Omron Sysmac Studio project Matching_Code_10 (Sysmac Studio 1.54.0.64019, StandardProject)
(* update 6_7 / have modify the res for fully reset home flag *)

# Controller new_Controller_0: NX1P2-1140DT version 1.18
Units and slaves: Node47 : MADLN05BE (E002); Node72 : MADLN05BE (E001); Node73 : MADLN05BE (E003)
Axis MC_Axis1, settings changed from default: AxisType=ServoType, UnitsConversion=EnumElement5, UnitsNumerator=8388608, UnitsDenominator=36, MaxVelocity=500, MaxJogVelocity=360, SoftwareLimitMode=ValidForSpecifiedValueImmediateStop, PositiveSoftwareLimit=75, NegativeSoftwareLimit=-29.2, OriginInputMode=EXT, StartDirection=NegativeDirection, OriginInputDetectionDirection=NegativeDirection, HomingVelocity=100, HomingApproachVelocity=10, HomingAcceleration=10, HomingDeceleration=20
Axis MC_Axis2, settings changed from default: AxisNumber=1, AxisType=ServoType, UnitsConversion=EnumElement5, UnitsNumerator=8388608, UnitsDenominator=36, MaxVelocity=500, MaxJogVelocity=360, SoftwareLimitMode=ValidForSpecifiedValueImmediateStop, PositiveSoftwareLimit=75, NegativeSoftwareLimit=-29.2
Axis MC_Axis3, settings changed from default: AxisNumber=2, AxisType=ServoType, UnitsConversion=EnumElement5, UnitsNumerator=8388608, UnitsDenominator=36, MaxVelocity=500, MaxJogVelocity=360, SoftwareLimitMode=ValidForSpecifiedValueDecreaseStop, PositiveSoftwareLimit=29.2, NegativeSoftwareLimit=-75
Task PrimaryTask (priority 4, period or condition 4000): Program0

TYPE InforRobot : STRUCT
    e : LREAL;
    rf : LREAL;
    re : LREAL;
    f : LREAL;
END_STRUCT END_TYPE
TYPE Input_Position : STRUCT
    X : LREAL;
    Y : LREAL;
    Z : LREAL;
END_STRUCT END_TYPE
TYPE Angle_Theta : STRUCT
    Theta1 : LREAL;
    Theta2 : LREAL;
    Theta3 : LREAL;
END_STRUCT END_TYPE
TYPE Bool_Theta : STRUCT
    Motor_Theta1 : REAL;
    Motor_Theta2 : REAL;
    Motor_Theta3 : REAL;
END_STRUCT END_TYPE
TYPE Speed_Theta : STRUCT
    Speed_Theta1 : REAL;
    Speed_Theta2 : REAL;
    Speed_Theta3 : REAL;
END_STRUCT END_TYPE
TYPE Workspace : STRUCT
    X_Min : REAL;
    X_Max : REAL;
    Y_Min : REAL;
    Y_Max : REAL;
    Z_Min : REAL;
    Z_Max : REAL;
END_STRUCT END_TYPE
TYPE From_pc : STRUCT
    commandID : INT;
    argument_number : INT;
    argument_x : ARRAY[0..6] OF real;
    argument_y : ARRAY[0..6] OF real;
    argument_z : ARRAY[0..6] OF real;
    argument_time : ARRAY[0..6] OF real;
    argument_e : ARRAY[0..6] OF int;
    bit_doing : INT;
END_STRUCT END_TYPE
TYPE From_plc : STRUCT
    pos_angular : ARRAY[0..2] OF REAL;
    pos_EE : ARRAY[0..6] OF REAL;
    task_doing : INT;
    task_state : INT;
    Total_Time_Estimate : ARRAY[0..6] OF REAL;
END_STRUCT END_TYPE

VAR_GLOBAL CONSTANT
    MC_Axis1 : _sAXIS_REF;  (* at MC://_MC_AX[0] *)
    MC_Axis2 : _sAXIS_REF;  (* at MC://_MC_AX[1] *)
    MC_Axis3 : _sAXIS_REF;  (* at MC://_MC_AX[2] *)
END_VAR
VAR_GLOBAL
    Out_Test0 : LREAL;
    Out_TestAngle1 : LREAL;
    Out_TestAngle2 : LREAL;
    Out_TestAngle3 : LREAL;
    MyHomingPara : _sHOMING_REF;
    Home_Axis1 : BOOL;  (* at BuiltInIO://cpu/#0/Input_Bit_00 *)
    Home_Axis2 : BOOL;  (* at BuiltInIO://cpu/#0/Input_Bit_01 *)
    Home_Axis3 : BOOL;  (* at BuiltInIO://cpu/#0/Input_Bit_02 *)
    Home_Lamp1 : BOOL;  (* at BuiltInIO://cpu/#0/Output_Bit_00 *)
    Home_Lamp2 : BOOL;  (* at BuiltInIO://cpu/#0/Output_Bit_01 *)
    Home_Lamp3 : BOOL;  (* at BuiltInIO://cpu/#0/Output_Bit_02 *)
    Out_Done_Inter : BOOL;
    pc_package : From_pc;  (* published *)
    plc_package : From_plc;  (* published *)
    Pump_Out : BOOL;  (* at BuiltInIO://cpu/#0/Output_Bit_03 *)
    Mc_On_Btn : BOOL;  (* at BuiltInIO://cpu/#0/Input_Bit_03 *)
    Res_Err_Btn : BOOL;  (* at BuiltInIO://cpu/#0/Input_Bit_04 *)
    Valve_Out : BOOL;  (* at BuiltInIO://cpu/#0/Output_Bit_04 *)
    ICV_t : ARRAY[0..6] OF Lreal;
    Start_Home_Flag : BOOL;
    Home_Done_Flag1 : BOOL;
    Home_Done_Flag2 : BOOL;
    Home_Done_Flag3 : BOOL;
END_VAR

PROGRAM Program0
VAR
    Pw_servo_on : BOOL := False;
    MC_Move_Abs : BOOL;
    Pw_Power_0 : MC_Power;
    Pw_Power_1 : MC_Power;
    Pw_Power_2 : MC_Power;
    MC_Home_Ext : BOOL;  (* toggle 1 *)
    MC_Home_Delta_0 : MC_Home_Delta;
    Calib_Abs1 : MC_MoveAbsolute;
    Calib_Abs2 : MC_MoveAbsolute;
    Calib_Abs3 : MC_MoveAbsolute;
    Home_test_1 : MC_Home;
    Home_test_2 : MC_Home;
    Home_test_3 : MC_Home;
    Move_abs_0 : MC_MoveAbsolute;
    Move_abs_1 : MC_MoveAbsolute;
    Move_abs_2 : MC_MoveAbsolute;
    X_cal : LREAL;
    Y_cal : LREAL;
    Z_cal : LREAL;
    pos_angular : LREAL;
    Exe_Inter1 : BOOL;
    Exe_Inter2 : BOOL;
    Count1 : UINT;
    Count2 : UINT;
    Goto_Abs : Goto_Absolute;
    when_it_turn2 : BOOL;
    Goto_abs_x : LREAL;
    Goto_abs_y : LREAL;
    Goto_abs_z : LREAL;
    another3 : BOOL;
    Count3 : UINT;
    another4 : BOOL;
    Count4 : UINT;
    MC_Inter_Curve_Vel_0 : MC_Inter_Curve_Vel;
    MC_Inter_Curve_Vel_1 : MC_Inter_Curve_Vel;
    MC_Inter_Curve_Vel_2 : MC_Inter_Curve_Vel;
    MC_Inter_Curve_Vel_3 : MC_Inter_Curve_Vel;
    MC_Inter_Curve_Vel_4 : MC_Inter_Curve_Vel;
    MC_Inter_Curve_Vel_5 : MC_Inter_Curve_Vel;
    ICV_Start_NewTurn : BOOL;  (* Set 1 until ICV_Blend_done_2 *)
    ICV_Blend_Done_0 : BOOL;  (* Exe auto turn zero right after finish the blend, and blend will true right after *)
    ICV_Blend_Done_1 : BOOL;
    ICV_Blend_Done_2 : BOOL;
    ICV_Blend_Done_3 : BOOL;
    ICV_Blend_Done_4 : BOOL;
    ICV_Blend_Done_5 : BOOL;
    ICV_Vend_0 : LREAL;  (* Err_IK must reset manual *)
    ICV_Vend_1 : LREAL;
    ICV_Vend_2 : LREAL;
    ICV_Vend_3 : LREAL;
    ICV_Vend_4 : LREAL;
    ICV_Vend_5 : LREAL;
    ICV_Vmax : LREAL := 300;  (* 300 *)
    ICV_Amax : LREAL := 1000;  (* 1000 *)
    ICV_Dmax : LREAL := 1000;  (* 1000 *)
    Pump_Ext : BOOL;
    ICV_Pos_E : ARRAY[0..6] OF Int;
    ICV_Pos_X : ARRAY[0..6] OF Lreal;
    ICV_Pos_Y : ARRAY[0..6] OF Lreal;
    ICV_Pos_Z : ARRAY[0..6] OF Lreal;
    i1 : INT;
    MC_Goto_Abs : BOOL;  (* Set 1 until it done *)
    Fwk_Calc_OutX : REAL;
    Fwk_Calc_OutY : REAL;
    Fwk_Calc_OutZ : REAL;
    Moveto_Intermediary : MC_MoveAbsolute;
    Moveto_Midpoint : MC_MoveAbsolute;
    Moveto_Midpoint_1 : MC_MoveAbsolute;
    Moveto_Midpoint_2 : MC_MoveAbsolute;
    Moveto_Midpoint_3 : MC_MoveAbsolute;
    Home_Done : BOOL;
    Home_Error : BOOL;
    Goto_Abs_Error : BOOL;
    Pump_Res : BOOL;
    MC_ICV_Err : BOOL;
    MC_Stop1 : MC_Stop;
    MC_Stop2 : MC_Stop;
    MC_Stop3 : MC_Stop;
    MC_RES_DB1 : MC_Reset;
    MC_RES_DB2 : MC_Reset;
    MC_RES_DB3 : MC_Reset;
    Comment : BOOL;
    Mc_On_Btn_Flag : BOOL;
    Check_IK : BOOL;
    Goto_Abs2 : Goto_Absolute;
    Goto_Abs2_Exe : BOOL;
    Goto_Abs2_Done : BOOL;
    Out_TestAngle1_tmp : LREAL;
    Out_TestAngle2_tmp : LREAL;
    Out_TestAngle3_tmp : LREAL;
    Out_TestAngle10 : LREAL;
    Out_TestAngle20 : LREAL;
    Out_TestAngle30 : LREAL;
    Stop1 : MC_Power;
    MC_Stop4 : MC_Stop;
    MC_Stop5 : MC_Stop;
    MC_Stop6 : MC_Stop;
    Comment0 : BOOL;
    MC_Inter_Curve_Vel_6 : MC_Inter_Curve_Vel;
    ICV_Blend_Done_6 : BOOL;
    ICV_Vend_6 : LREAL;
    Current_Step : INT;
    Axis1_test : LREAL;
    Axis2_test : LREAL;
    Axis3_test : LREAL;
    fb_PumpTimer : TP;
    Var_Timer_IN : BOOL;
    ICV_t0 : LREAL;
    ICV_t1 : LREAL;
    ICV_t2 : LREAL;
    ICV_t3 : LREAL;
    ICV_t4 : LREAL;
    ICV_t5 : LREAL;
    Timing_for_EEF : TIME;
    i_t : INT;
    Mem_ICV_t5 : LREAL;
    k_t : LREAL;
    Pos_calib1 : LREAL;
    Pos_calib2 : LREAL;
    Pos_calib3 : LREAL;
END_VAR
VAR_EXTERNAL
    Out_Test0 : LREAL;
    Out_TestAngle1 : LREAL;
    Out_TestAngle2 : LREAL;
    Out_TestAngle3 : LREAL;
END_VAR
VAR_EXTERNAL CONSTANT
    MC_Axis1 : _sAXIS_REF;
    MC_Axis2 : _sAXIS_REF;
    MC_Axis3 : _sAXIS_REF;
END_VAR
VAR_EXTERNAL
    Home_Axis2 : BOOL;
    Home_Axis3 : BOOL;
    Out_Done_Inter : BOOL;
    plc_package : From_plc;
    pc_package : From_pc;
    Pump_Out : BOOL;
    Home_Axis1 : BOOL;
    Mc_On_Btn : BOOL;
    Res_Err_Btn : BOOL;
    Valve_Out : BOOL;
    ICV_t : ARRAY[0..6] OF Lreal;
    Start_Home_Flag : BOOL;
    Home_Done_Flag1 : BOOL;
    Home_Done_Flag2 : BOOL;
    Home_Done_Flag3 : BOOL;
END_VAR
VAR
    _p1 : BOOL;
    _t2 : BOOL;
    _t3 : BOOL;
END_VAR

(* Section Section0: ladder, written here as Structured Text *)

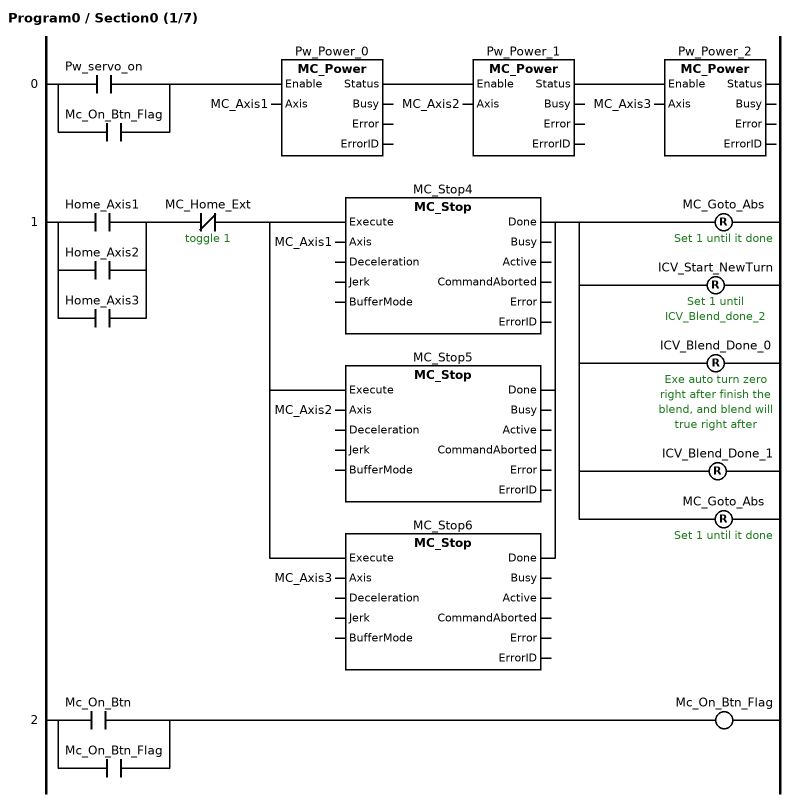
(* Rung 0 *)
Pw_Power_0(Enable := Pw_servo_on OR Mc_On_Btn_Flag, Axis := MC_Axis1);
Pw_Power_1(Enable := Pw_Power_0.Status, Axis := MC_Axis2);
Pw_Power_2(Enable := Pw_Power_1.Status, Axis := MC_Axis3);
(* Rung 1 *)
_p1 := (Home_Axis1 OR Home_Axis2 OR Home_Axis3) AND NOT MC_Home_Ext;
MC_Stop4(Execute := _p1, Axis := MC_Axis1);
MC_Stop5(Execute := _p1, Axis := MC_Axis2);
MC_Stop6(Execute := _p1, Axis := MC_Axis3);
IF MC_Stop4.Done OR MC_Stop5.Done OR MC_Stop6.Done THEN
    MC_Goto_Abs := FALSE;
    ICV_Start_NewTurn := FALSE;
    ICV_Blend_Done_0 := FALSE;
    ICV_Blend_Done_1 := FALSE;
    MC_Goto_Abs := FALSE;
END_IF;
(* Rung 2 *)
Mc_On_Btn_Flag := Mc_On_Btn OR Mc_On_Btn_Flag;

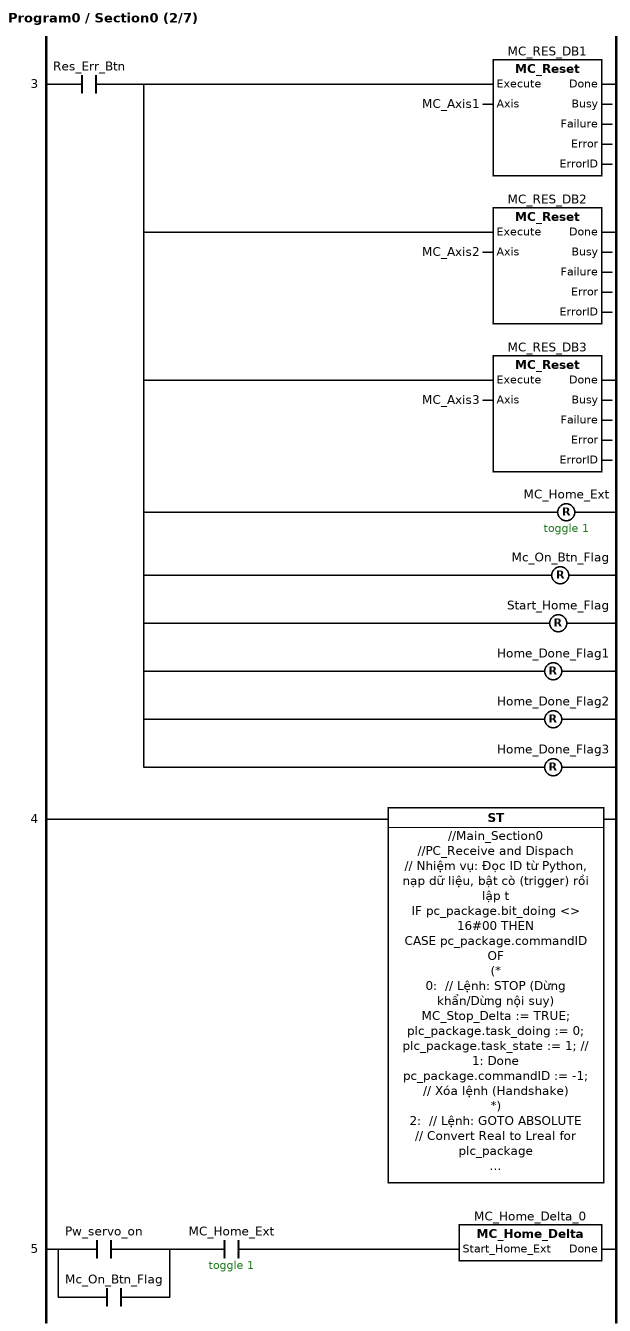
(* Rung 3 *)
MC_RES_DB1(Execute := Res_Err_Btn, Axis := MC_Axis1);
MC_RES_DB2(Execute := Res_Err_Btn, Axis := MC_Axis2);
MC_RES_DB3(Execute := Res_Err_Btn, Axis := MC_Axis3);
IF Res_Err_Btn THEN
    MC_Home_Ext := FALSE;
    Mc_On_Btn_Flag := FALSE;
    Start_Home_Flag := FALSE;
    Home_Done_Flag1 := FALSE;
    Home_Done_Flag2 := FALSE;
    Home_Done_Flag3 := FALSE;
END_IF;
(* Rung 4 *)
//Main_Section0 
//PC_Receive and Dispach
// Nhiệm vụ: Đọc ID từ Python, nạp dữ liệu, bật cò (trigger) rồi lập tức xóa ID

IF pc_package.bit_doing <> 16#00 THEN
CASE pc_package.commandID OF
  (*  
0:  // Lệnh: STOP (Dừng khẩn/Dừng nội suy)
	        MC_Stop_Delta := TRUE;
	        
	        plc_package.task_doing := 0;
	        plc_package.task_state := 1; // 1: Done
	        pc_package.commandID := -1;  // Xóa lệnh (Handshake)
			*)
    2:  // Lệnh: GOTO ABSOLUTE
		// Convert Real to Lreal for plc_package
		Goto_abs_x:= REAL_TO_LREAL(pc_package.argument_x[0]);
		Goto_abs_y := REAL_TO_LREAL(pc_package.argument_y[0]);
		Goto_abs_z:= REAL_TO_LREAL(pc_package.argument_z[0]);
        
        MC_Goto_Abs := TRUE;         // Bật cò chạy
        plc_package.task_doing := 2;
        plc_package.task_state := 2; // 2: Busy
        pc_package.commandID := -1;

    3:  // Lệnh: GO TRAJECTORY (Chạy quỹ đạo theo mảng tọa độ)
        ICV_Start_NewTurn := TRUE; //auto turn off
        FOR i1 := 0 TO 6 DO
			ICV_Pos_X[i1] := REAL_TO_LREAL(pc_package.argument_x[i1]);
			ICV_Pos_Y[i1] := REAL_TO_LREAL(pc_package.argument_y[i1]);
			ICV_Pos_Z[i1] := REAL_TO_LREAL(pc_package.argument_z[i1]);
			ICV_Pos_E[i1] := pc_package.argument_e[i1];
		END_FOR;
        plc_package.task_doing := 3;
        plc_package.task_state := 2; // Busy
        pc_package.commandID := -1;

    4:  // Lệnh: HOME CALIBRATION (Tìm gốc)
        MC_Home_Ext := TRUE;
        
        plc_package.task_doing := 4;
        plc_package.task_state := 2; // Busy
        pc_package.commandID := -1;

    5:  // Lệnh: PICK (Hút vật)
        Pump_Ext := TRUE;
        
        plc_package.task_doing := 5;
        plc_package.task_state := 1; // 1: Done (Do bật bơm là xong ngay)
        pc_package.commandID := -1;

    6:  // Lệnh: RELEASE (Nhả vật)
        Pump_Ext := FALSE;
        
        plc_package.task_doing := 6;
        plc_package.task_state := 1; // Done
        pc_package.commandID := -1;
		END_CASE;
pc_package.bit_doing :=16#00;
END_IF;
(* Rung 5 *)
MC_Home_Delta_0(Start_Home_Ext := (Pw_servo_on OR Mc_On_Btn_Flag) AND MC_Home_Ext);

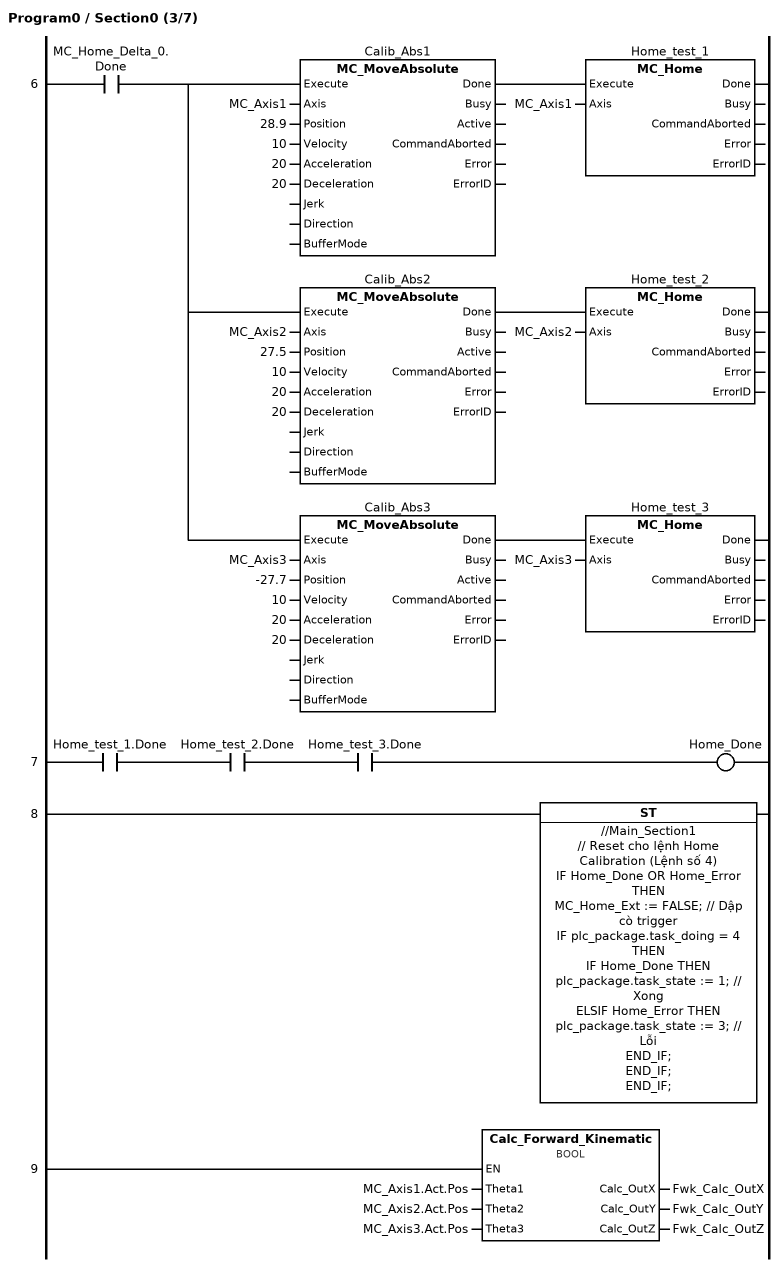
(* Rung 6 *)
Calib_Abs1(Execute := MC_Home_Delta_0.Done, Axis := MC_Axis1, Position := 28.9, Velocity := 10, Acceleration := 20, Deceleration := 20);
Home_test_1(Execute := Calib_Abs1.Done, Axis := MC_Axis1);
Calib_Abs2(Execute := MC_Home_Delta_0.Done, Axis := MC_Axis2, Position := 27.5, Velocity := 10, Acceleration := 20, Deceleration := 20);
Home_test_2(Execute := Calib_Abs2.Done, Axis := MC_Axis2);
Calib_Abs3(Execute := MC_Home_Delta_0.Done, Axis := MC_Axis3, Position := -27.7, Velocity := 10, Acceleration := 20, Deceleration := 20);
Home_test_3(Execute := Calib_Abs3.Done, Axis := MC_Axis3);
(* Rung 7 *)
Home_Done := Home_test_1.Done AND Home_test_2.Done AND Home_test_3.Done;
(* Rung 8 *)
//Main_Section1 
// Reset cho lệnh Home Calibration (Lệnh số 4)
IF Home_Done OR Home_Error THEN
 
    MC_Home_Ext := FALSE; // Dập cò trigger
	
    IF plc_package.task_doing = 4 THEN
        IF Home_Done THEN
            plc_package.task_state := 1; // Xong
        ELSIF Home_Error THEN
            plc_package.task_state := 3; // Lỗi
        END_IF;
    END_IF;
    
END_IF;
(* Rung 9 *)
_t2 := Calc_Forward_Kinematic(Theta1 := MC_Axis1.Act.Pos, Theta2 := MC_Axis2.Act.Pos, Theta3 := MC_Axis3.Act.Pos, Calc_OutX => Fwk_Calc_OutX, Calc_OutY => Fwk_Calc_OutY, Calc_OutZ => Fwk_Calc_OutZ);

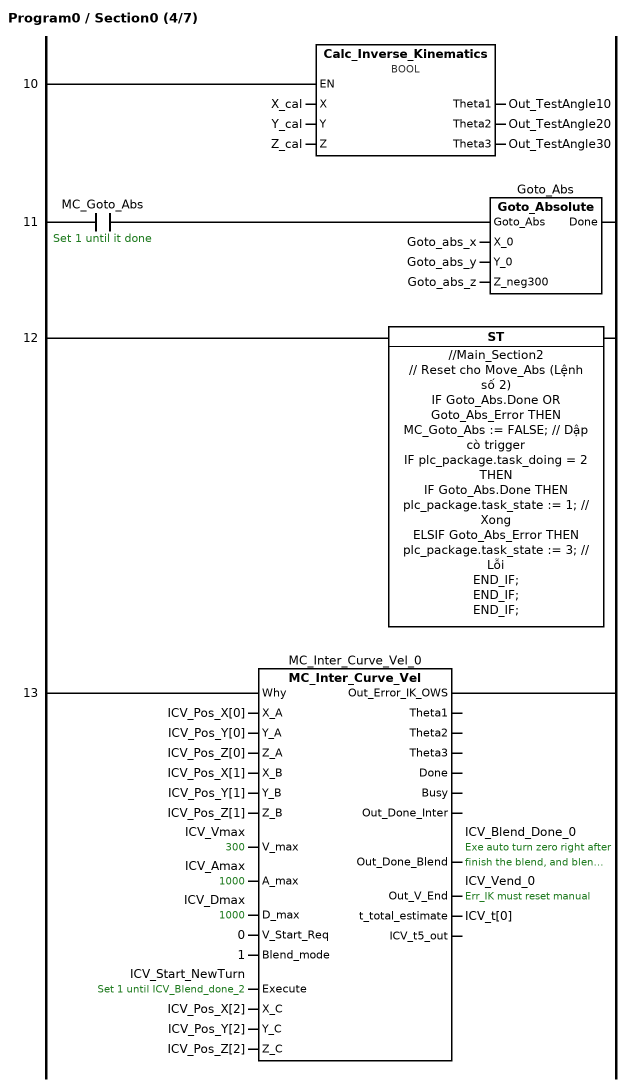
(* Rung 10 *)
_t3 := Calc_Inverse_Kinematics(X := X_cal, Y := Y_cal, Z := Z_cal, Theta1 => Out_TestAngle10, Theta2 => Out_TestAngle20, Theta3 => Out_TestAngle30);
(* Rung 11 *)
Goto_Abs(Goto_Abs := MC_Goto_Abs, X_0 := Goto_abs_x, Y_0 := Goto_abs_y, Z_neg300 := Goto_abs_z);
(* Rung 12 *)
//Main_Section2
// Reset cho Move_Abs (Lệnh số 2)
IF Goto_Abs.Done OR Goto_Abs_Error THEN
 
    MC_Goto_Abs := FALSE; // Dập cò trigger
	
    IF plc_package.task_doing = 2 THEN
        IF Goto_Abs.Done THEN
            plc_package.task_state := 1; // Xong
        ELSIF Goto_Abs_Error THEN
            plc_package.task_state := 3; // Lỗi
        END_IF;
    END_IF;
    
END_IF;
(* Rung 13 *)
MC_Inter_Curve_Vel_0(Why := TRUE, X_A := ICV_Pos_X[0], Y_A := ICV_Pos_Y[0], Z_A := ICV_Pos_Z[0], X_B := ICV_Pos_X[1], Y_B := ICV_Pos_Y[1], Z_B := ICV_Pos_Z[1], V_max := ICV_Vmax, A_max := ICV_Amax, D_max := ICV_Dmax, V_Start_Req := 0, Blend_mode := 1, Execute := ICV_Start_NewTurn, X_C := ICV_Pos_X[2], Y_C := ICV_Pos_Y[2], Z_C := ICV_Pos_Z[2], Out_Done_Blend => ICV_Blend_Done_0, Out_V_End => ICV_Vend_0, t_total_estimate => ICV_t[0]);

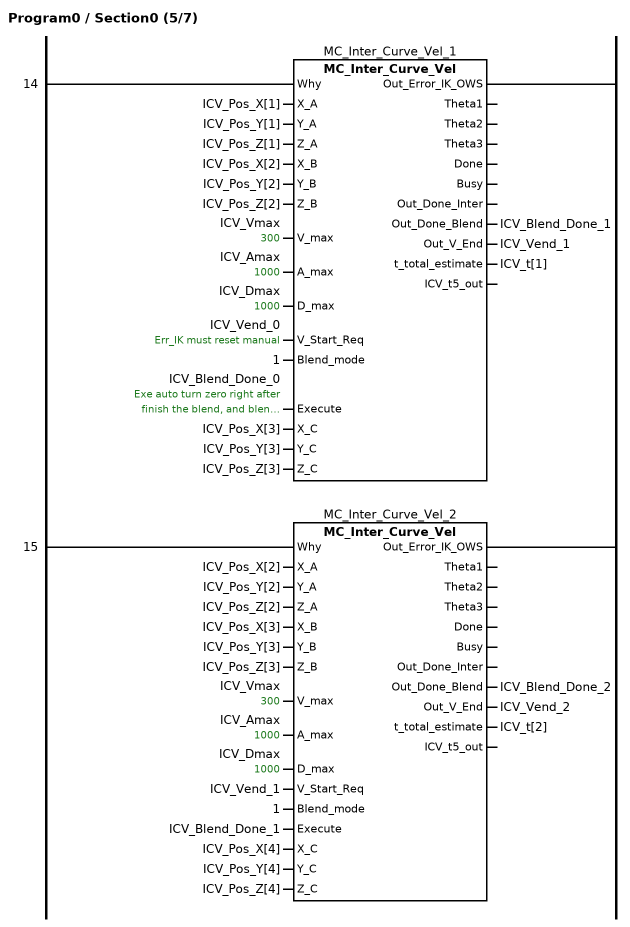
(* Rung 14 *)
MC_Inter_Curve_Vel_1(Why := TRUE, X_A := ICV_Pos_X[1], Y_A := ICV_Pos_Y[1], Z_A := ICV_Pos_Z[1], X_B := ICV_Pos_X[2], Y_B := ICV_Pos_Y[2], Z_B := ICV_Pos_Z[2], V_max := ICV_Vmax, A_max := ICV_Amax, D_max := ICV_Dmax, V_Start_Req := ICV_Vend_0, Blend_mode := 1, Execute := ICV_Blend_Done_0, X_C := ICV_Pos_X[3], Y_C := ICV_Pos_Y[3], Z_C := ICV_Pos_Z[3], Out_Done_Blend => ICV_Blend_Done_1, Out_V_End => ICV_Vend_1, t_total_estimate => ICV_t[1]);
(* Rung 15 *)
MC_Inter_Curve_Vel_2(Why := TRUE, X_A := ICV_Pos_X[2], Y_A := ICV_Pos_Y[2], Z_A := ICV_Pos_Z[2], X_B := ICV_Pos_X[3], Y_B := ICV_Pos_Y[3], Z_B := ICV_Pos_Z[3], V_max := ICV_Vmax, A_max := ICV_Amax, D_max := ICV_Dmax, V_Start_Req := ICV_Vend_1, Blend_mode := 1, Execute := ICV_Blend_Done_1, X_C := ICV_Pos_X[4], Y_C := ICV_Pos_Y[4], Z_C := ICV_Pos_Z[4], Out_Done_Blend => ICV_Blend_Done_2, Out_V_End => ICV_Vend_2, t_total_estimate => ICV_t[2]);

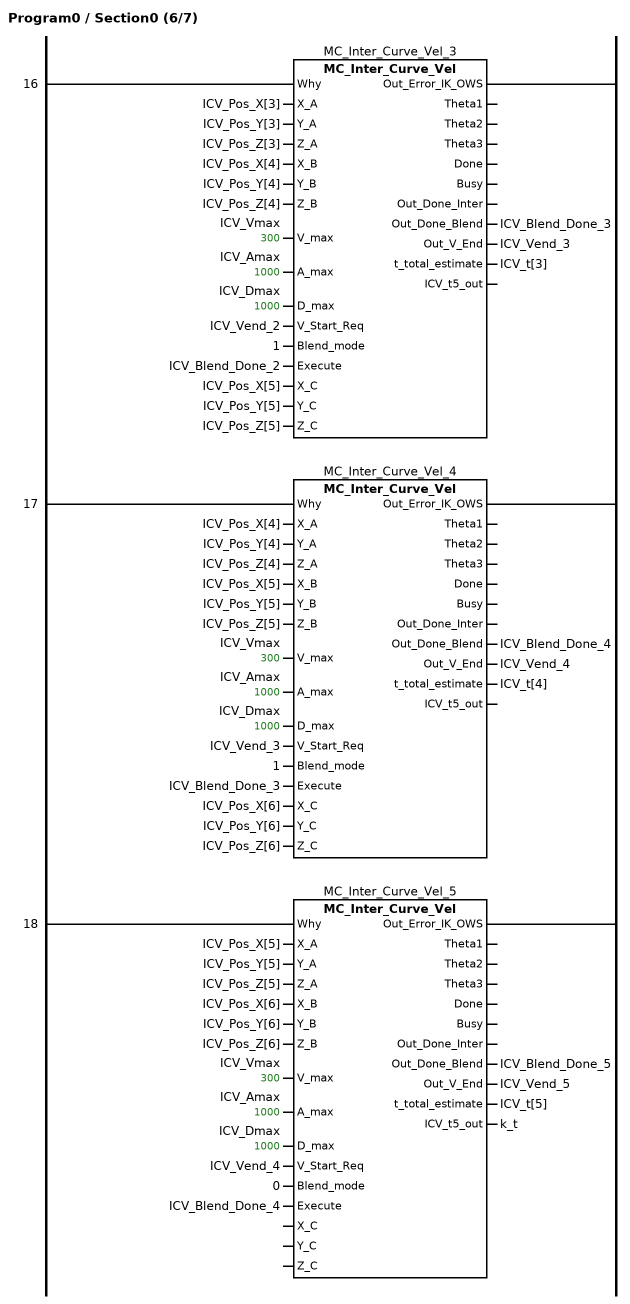
(* Rung 16 *)
MC_Inter_Curve_Vel_3(Why := TRUE, X_A := ICV_Pos_X[3], Y_A := ICV_Pos_Y[3], Z_A := ICV_Pos_Z[3], X_B := ICV_Pos_X[4], Y_B := ICV_Pos_Y[4], Z_B := ICV_Pos_Z[4], V_max := ICV_Vmax, A_max := ICV_Amax, D_max := ICV_Dmax, V_Start_Req := ICV_Vend_2, Blend_mode := 1, Execute := ICV_Blend_Done_2, X_C := ICV_Pos_X[5], Y_C := ICV_Pos_Y[5], Z_C := ICV_Pos_Z[5], Out_Done_Blend => ICV_Blend_Done_3, Out_V_End => ICV_Vend_3, t_total_estimate => ICV_t[3]);
(* Rung 17 *)
MC_Inter_Curve_Vel_4(Why := TRUE, X_A := ICV_Pos_X[4], Y_A := ICV_Pos_Y[4], Z_A := ICV_Pos_Z[4], X_B := ICV_Pos_X[5], Y_B := ICV_Pos_Y[5], Z_B := ICV_Pos_Z[5], V_max := ICV_Vmax, A_max := ICV_Amax, D_max := ICV_Dmax, V_Start_Req := ICV_Vend_3, Blend_mode := 1, Execute := ICV_Blend_Done_3, X_C := ICV_Pos_X[6], Y_C := ICV_Pos_Y[6], Z_C := ICV_Pos_Z[6], Out_Done_Blend => ICV_Blend_Done_4, Out_V_End => ICV_Vend_4, t_total_estimate => ICV_t[4]);
(* Rung 18 *)
MC_Inter_Curve_Vel_5(Why := TRUE, X_A := ICV_Pos_X[5], Y_A := ICV_Pos_Y[5], Z_A := ICV_Pos_Z[5], X_B := ICV_Pos_X[6], Y_B := ICV_Pos_Y[6], Z_B := ICV_Pos_Z[6], V_max := ICV_Vmax, A_max := ICV_Amax, D_max := ICV_Dmax, V_Start_Req := ICV_Vend_4, Blend_mode := 0, Execute := ICV_Blend_Done_4, Out_Done_Blend => ICV_Blend_Done_5, Out_V_End => ICV_Vend_5, t_total_estimate => ICV_t[5], ICV_t5_out => k_t);

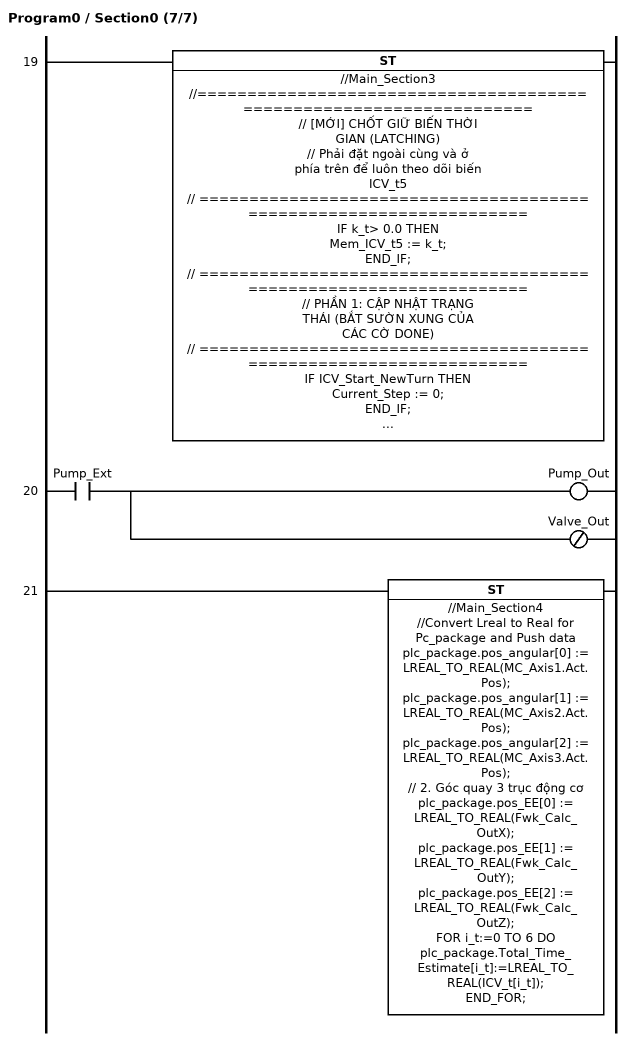
(* Rung 19 *)
//Main_Section3
//=========================================================================
// [MỚI] CHỐT GIỮ BIẾN THỜI GIAN (LATCHING)
// Phải đặt ngoài cùng và ở phía trên để luôn theo dõi biến ICV_t5
// =========================================================================
IF k_t> 0.0 THEN
    Mem_ICV_t5 := k_t;
END_IF;

// =========================================================================
// PHẦN 1: CẬP NHẬT TRẠNG THÁI (BẮT SƯỜN XUNG CỦA CÁC CỜ DONE)
// =========================================================================
IF ICV_Start_NewTurn THEN
    Current_Step := 0;
END_IF;

IF ICV_Blend_Done_0 THEN Current_Step := 1; END_IF;
IF ICV_Blend_Done_1 THEN Current_Step := 2; END_IF;
IF ICV_Blend_Done_2 THEN Current_Step := 3; END_IF;
IF ICV_Blend_Done_3 THEN Current_Step := 4; END_IF;
IF ICV_Blend_Done_4 THEN Current_Step := 5; END_IF;
IF ICV_Blend_Done_5 THEN Current_Step := 6; END_IF;

// =========================================================================
// PHẦN 2: CHUẨN BỊ TÍN HIỆU VÀ KÍCH HOẠT TIMER
// =========================================================================
Var_Timer_IN := FALSE; 

// Chỉ kích hoạt cờ IN khi đang ở Step 5
IF (Current_Step = 5) THEN
    Var_Timer_IN := TRUE; 
END_IF;

// Tính toán thời gian (t) dùng biến đã Latch: Mem_ICV_t5 với hệ số 0.7 (70%)
Timing_for_EEF := NanoSecToTime(LREAL_TO_LINT(0.5 * Mem_ICV_t5 * 1000000000.0));

// Gọi khối Timer chạy ngầm (Giả định là TON)
fb_PumpTimer(
    IN := Var_Timer_IN, 
    PT := Timing_for_EEF 
);

// =========================================================================
// PHẦN 3: ĐIỀU KHIỂN BƠM (STATE MACHINE)
// =========================================================================
CASE Current_Step OF
    0: Pump_Ext := (ICV_Pos_E[0] = 1);
    1: Pump_Ext := (ICV_Pos_E[1] = 1);
    2: Pump_Ext := (ICV_Pos_E[2] = 1);
    3: Pump_Ext := (ICV_Pos_E[3] = 1);
    4: Pump_Ext := (ICV_Pos_E[4] = 1);
    
    5: 
        // Bơm bật nếu mảng lệnh cho phép (=1) VÀ Timer chưa đếm xong 70% thời gian.
        // Khi TON đếm đủ giờ, .Q = TRUE -> NOT .Q = FALSE -> Bơm ngắt.
        // Nếu khối fb_PumpTimer của bạn là loại TP (Pulse Timer), hãy đổi thành: AND fb_PumpTimer.Q;
        Pump_Ext := (ICV_Pos_E[5] = 1) AND fb_PumpTimer.Q; 
        
    6: 
        Pump_Ext := FALSE;
        
ELSE 
    Pump_Ext := FALSE;
END_CASE;
(* Rung 20 *)
Pump_Out := Pump_Ext;
Valve_Out := NOT Pump_Ext;
(* Rung 21 *)
//Main_Section4
//Convert Lreal to Real for Pc_package and Push data
plc_package.pos_angular[0] := LREAL_TO_REAL(MC_Axis1.Act.Pos);
plc_package.pos_angular[1] := LREAL_TO_REAL(MC_Axis2.Act.Pos);
plc_package.pos_angular[2] := LREAL_TO_REAL(MC_Axis3.Act.Pos);

// 2. Góc quay 3 trục động cơ
plc_package.pos_EE[0] := LREAL_TO_REAL(Fwk_Calc_OutX); 
plc_package.pos_EE[1] := LREAL_TO_REAL(Fwk_Calc_OutY); 
plc_package.pos_EE[2] := LREAL_TO_REAL(Fwk_Calc_OutZ);

FOR i_t:=0 TO 6 DO
	plc_package.Total_Time_Estimate[i_t]:=LREAL_TO_REAL(ICV_t[i_t]);
END_FOR;
END_PROGRAM

FUNCTION Calc_Inverse_Kinematics : BOOL
VAR CONSTANT
    Cos120 : LREAL := -0.5;
    Sin120 : LREAL := 0.8660254037844386;
END_VAR
VAR
    tmp_Theta1 : LREAL;
    tmp_Theta2 : LREAL;
    tmp_Theta3 : LREAL;
    rotate_X2 : LREAL;
    rotate_Y2 : LREAL;
    rotate_X3 : LREAL;
    rotate_Y3 : LREAL;
END_VAR
VAR CONSTANT
    rf : LREAL := 346.4;
    re : LREAL := 86.6;
    f : LREAL := 140;
    e : LREAL := 315;
END_VAR
VAR
    Out_Error_IK : BOOL;
END_VAR
VAR_INPUT
    X : LREAL;
    Y : LREAL;
    Z : LREAL;
END_VAR
VAR_OUTPUT
    Theta1 : LREAL;
    Theta2 : LREAL;
    Theta3 : LREAL;
END_VAR
// Khởi tạo lại cờ báo lỗi ở mỗi đầu chu kỳ quét (Primary Task)
Out_Error_IK := FALSE;

// -----------------------------------------------------------------------
// TÍNH TOÁN THETA 1 (Cánh tay 1 - Không xoay trục)
// -----------------------------------------------------------------------
Calc_Inverse_Kinematics := Calc_Angles_YZ(
    X0 := X, 
    Y0 := Y, 
    Z0 := Z,
    OutTheta => tmp_Theta1
);

	
// [TỐI ƯU B] Xử lý lỗi an toàn: Nếu tính toán IK thất bại (Tọa độ ngoài tầm với)
IF Calc_Inverse_Kinematics = TRUE  OR tmp_Theta1 <-20 THEN
    Out_Error_IK := TRUE; // Bật cờ báo lỗi ra hệ thống
    RETURN;               // Ngắt tính toán ngay lập tức
END_IF;

// [TỐI ƯU A] Truyền thẳng giá trị LREAL nguyên bản xuống Servo, BỎ HÀM ROUND
Theta1 := tmp_Theta1;


// -----------------------------------------------------------------------
// TÍNH TOÁN THETA 2 (Cánh tay 2 - Xoay hệ tọa độ đi -120 độ)
// -----------------------------------------------------------------------
rotate_X2 := X * Cos120 + Y * Sin120;
rotate_Y2 := Y * Cos120 - X * Sin120;

Calc_Inverse_Kinematics := Calc_Angles_YZ(
    X0 := rotate_X2, 
    Y0 := rotate_Y2, 
    Z0 := Z,
    OutTheta => tmp_Theta2
);

IF Calc_Inverse_Kinematics = TRUE OR tmp_Theta2 <-20 THEN
    Out_Error_IK := TRUE;
    RETURN;
END_IF;

Theta2 := tmp_Theta2;


// -----------------------------------------------------------------------
// TÍNH TOÁN THETA 3 (Cánh tay 3 - Xoay hệ tọa độ đi +120 độ)
// -----------------------------------------------------------------------
rotate_X3 := X * Cos120 - Y * Sin120;
rotate_Y3 := Y * Cos120 + X * Sin120;

Calc_Inverse_Kinematics := Calc_Angles_YZ(
    X0 := rotate_X3, 
    Y0 := rotate_Y3, 
    Z0 := Z,
    OutTheta => tmp_Theta3
);

IF Calc_Inverse_Kinematics = TRUE OR tmp_Theta3*-1 >20 THEN
    Out_Error_IK := TRUE;
    RETURN;
END_IF;

Theta3 := tmp_Theta3*-1;
END_FUNCTION

FUNCTION Calc_Angles_YZ : BOOL  (* return true -> False in inverse calc *)
VAR
    tmp_y0 : LREAL;
    a : LREAL;
    b : LREAL;
    d : LREAL;
    yj : LREAL;
    zj : LREAL;
    y1 : LREAL;
    tmp_AnglePi : LREAL;
END_VAR
VAR CONSTANT
    Pi : LREAL := 3.141592653589793;
    Tan30 : LREAL := 0.5773502691896257;
    Base : LREAL := 346.4;
    EndEffector : LREAL := 86.6;
    Bicep : LREAL := 140;
    Forearm : LREAL := 315;
END_VAR
VAR_INPUT
    X0 : LREAL;
    Y0 : LREAL;
    Z0 : LREAL;
END_VAR
VAR_OUTPUT
    OutTheta : LREAL;
END_VAR
(*
// FUNCTION: Calc_Angles_YZ (Cal the inverse in 2D-space)
//All variants use Lreal to uttilize the precision of servo and syns all data

// [] Bẫy lỗi chia cho 0: Nếu tọa độ Z0 = 0 (End-effector nằm ngang với Base)
// Phép tính 'a' và 'b' bên dưới sẽ bị lỗi chia cho 0 làm CPU PLC báo lỗi (Major Fault)
*)
IF Z0 = 0.0 THEN
    Calc_Angles_YZ := TRUE; // turn Error true
    RETURN;
END_IF;

// Calc the Y1 and have temp_y0 (the prosition of the Y0 with Y1)
y1 := -0.5 * Tan30* Base;   // the point of edge of fix-triangle
tmp_y0 := Y0 - (0.5 *Tan30* EndEffector);  // the point of the edge of active-triagle

// we have ellbow (0,yj,zj) is contraint with:
//1. on a circle (0,y1,0) with R = bicep so (yj-y1)^2 + z_j^2 = bicep^2
//2. distance from End-effector (X0, tmp_y0,z0) equal the Forearm so
// X0^2 + (tmp_y0 - yj)^2 + (z-zj)^2 = forearm^2
// mathemitical tranformation we have linear function z with a and b bellow
// zj = a + b*yj => we have zj and we tranfer it to equation 1 and solve the two level function with yj
a := (X0*X0 + tmp_y0 * tmp_y0 + Z0 * Z0 + Bicep * Bicep - Forearm * Forearm - y1 * y1) / (2.0 * Z0);
b := (y1 - tmp_y0) / Z0;

// the delta of two level function with yj
d := - (a + b * y1) * (a + b * y1) + Bicep * (b * b * Bicep + Bicep);

// Kiểm tra xem điểm có tồn tại trong vùng không gian (Workspace) không
IF d < 0.0 THEN
    Calc_Angles_YZ := TRUE; // Trả về lỗi (Điểm không với tới được)
    RETURN;
END_IF;

yj := (y1 - a * b - SQRT(d)) / (b * b + 1.0);
zj := a + b * yj;

tmp_AnglePi := 0.0;
IF yj > y1 THEN
    tmp_AnglePi := 180.0;
END_IF;

// [TỐI ƯU 3] Bẫy lỗi chia cho 0 trong hàm tính góc ATAN
// Khi y1 = yj, phép chia (-zj / (y1 - yj)) sẽ gây lỗi PLC
IF (y1 - yj) = 0.0 THEN
    IF -zj >= 0.0 THEN
        OutTheta := 90.0 + tmp_AnglePi;
    ELSE
        OutTheta := -90.0 + tmp_AnglePi;
    END_IF;
ELSE
    // Tính góc Theta. Sử dụng hằng số '_pi' có sẵn của Sysmac Studio
    OutTheta := 180.0 * ATAN(-zj / (y1 - yj)) / Pi + tmp_AnglePi;
END_IF;

// Trả về FALSE khi tính toán thành công
Calc_Angles_YZ := FALSE;
RETURN;
END_FUNCTION

FUNCTION Calc_Forward_Kinematic : BOOL
VAR
    w : LREAL;
    Cos30 : LREAL := 0.8660254037844386;
    Pi : LREAL := 3.141592653589793;
    Tan30 : LREAL := 0.5773502691896257;
    Sin30 : LREAL := 0.5;
END_VAR
VAR CONSTANT
    Base : LREAL := 346.4;
    EndEffector : LREAL := 86.6;
    Bicep : LREAL := 140;
    Forearm : LREAL := 315;
END_VAR
VAR
    x_j1 : LREAL;
    y_j1 : LREAL;
    z_j1 : LREAL;
    x_j2 : LREAL;
    y_j2 : LREAL;
    z_j2 : LREAL;
    x_j3 : LREAL;
    y_j3 : LREAL;
    z_j3 : LREAL;
    r1 : LREAL;
    r2 : LREAL;
    r3 : LREAL;
    a1 : LREAL;
    a2 : LREAL;
    b1 : LREAL;
    b2 : LREAL;
    demon : LREAL;
    A_quad : LREAL;
    B_quad : LREAL;
    C_quad : LREAL;
    denom : LREAL;
    d : LREAL;
    t3 : LREAL;
    t2 : LREAL;
    t1 : LREAL;
    Calc_Forward_Kinematics : BOOL;
    OutX : LREAL;
    OutZ : LREAL;
    OutY : LREAL;
    D1_coeff : LREAL;
    A1_coeff : LREAL;
    B1_coeff : LREAL;
    C1_coeff : LREAL;
    A2_coeff : LREAL;
    B2_coeff : LREAL;
    C2_coeff : LREAL;
    D2_coeff : LREAL;
    det : LREAL;
END_VAR
VAR_INPUT
    Theta1 : LREAL;
    Theta2 : LREAL;
    Theta3 : LREAL;
END_VAR
VAR_OUTPUT
    Calc_OutX : REAL;
    Calc_OutY : REAL;
    Calc_OutZ : REAL;
END_VAR
VAR_EXTERNAL CONSTANT
    MC_Axis1 : _sAXIS_REF;
    MC_Axis2 : _sAXIS_REF;
    MC_Axis3 : _sAXIS_REF;
END_VAR
// =======================================================================
// FUNCTION: Calc_Forward_Kinematics (Tính toán động học thuận Robot Delta 3D)
// Trả về FALSE nếu tính toán thành công, TRUE nếu điểm nằm ngoài vùng làm việc
// =======================================================================
// LẤY GIÁ TRỊ GÓC THỰC TẾ (ACTUAL POSITION) TỪ ENCODER CỦA TRỤC
// =======================================================================
// Chuyển đổi các góc hiện tại từ Độ sang Radian
t1 := Theta1 * Pi / 180.0;
t2 := Theta2 * Pi / 180.0;
t3 := Theta3 * Pi / -180.0;

// Tính toán độ lệch tâm tương đối giữa Base và EndEffector
// (w chính là dịch tâm ngang từ gốc tọa độ đến khớp khuỷu tay nếu chiếu lên mặt phẳng XY)
w := 0.5 * Tan30 * (Base - EndEffector);

// =======================================================================
// BƯỚC 1: Tìm tọa độ không gian (x, y, z) của 3 khớp khuỷu tay (Elbow Joints)
// Hệ tọa độ tiêu chuẩn: Trục 1 nằm dọc theo phần âm của trục Y
// =======================================================================

// Trục 1 (Góc lệch 0 độ so với trục tính toán, xoay về -Y)
x_j1 := 0.0;
y_j1 := -(w + Bicep * COS(t1));
z_j1 := -Bicep * SIN(t1);

// Trục 2 (Xoay +120 độ)
x_j2 := (w + Bicep * COS(t2)) * Cos30;
y_j2 := (w + Bicep * COS(t2)) * Sin30;
z_j2 := -Bicep * SIN(t2);

// Trục 3 (Xoay -120 độ hoặc 240 độ)
x_j3 := -(w + Bicep * COS(t3)) * Cos30;
y_j3 := (w + Bicep * COS(t3)) * Sin30;
z_j3 := -Bicep * SIN(t3);

// =======================================================================
// BƯỚC 2: Giải hệ 3 phương trình mặt cầu có tâm tại các Elbow, bán kính Forearm
// =======================================================================

// =======================================================================
// BƯỚC 2: Giải hệ 3 phương trình mặt cầu (Dạng tổng quát, KHÔNG RÚT GỌN SAI)
// =======================================================================
// BƯỚC 2: Giải hệ 3 phương trình mặt cầu có tâm tại các Elbow (Phiên bản Tổng quát)
// =======================================================================

// Tính tổng bình phương tọa độ của các Elbow
r1 := y_j1 * y_j1 + z_j1 * z_j1;  // x_j1 = 0
r2 := x_j2 * x_j2 + y_j2 * y_j2 + z_j2 * z_j2;
r3 := x_j3 * x_j3 + y_j3 * y_j3 + z_j3 * z_j3;

// Thiết lập các hệ số cho hệ phương trình tuyến tính 2 ẩn (X, Y) theo tham số Z
// Dạng: 
// A1*X + B1*Y = D1 - C1*Z
// A2*X + B2*Y = D2 - C2*Z

A1_coeff := x_j2;                   // Thực chất là (x_j2 - x_j1) nhưng x_j1 = 0
B1_coeff := y_j2 - y_j1;
C1_coeff := z_j2 - z_j1;
D1_coeff := 0.5 * (r2 - r1);

A2_coeff := x_j3;                   // Thực chất là (x_j3 - x_j1) nhưng x_j1 = 0
B2_coeff := y_j3 - y_j1;
C2_coeff := z_j3 - z_j1;
D2_coeff := 0.5 * (r3 - r1);

// Tính định thức (Determinant) của hệ phương trình
det := (A1_coeff * B2_coeff) - (A2_coeff * B1_coeff);

// Bẫy lỗi: Hệ vô nghiệm (Chỉ xảy ra khi 3 khuỷu tay cùng nằm trên 1 đường thẳng)
IF det = 0.0 THEN
    Calc_Forward_Kinematics := TRUE; 
    RETURN;
END_IF;

// Sử dụng quy tắc Cramer để tìm a1, b1 (Cho X) và a2, b2 (Cho Y)
// Để biểu diễn: X0 = a1 + b1*Z0
a1 := (D1_coeff * B2_coeff - D2_coeff * B1_coeff) / det;
b1 := -(C1_coeff * B2_coeff - C2_coeff * B1_coeff) / det;

// Để biểu diễn: Y0 = a2 + b2*Z0
a2 := (A1_coeff * D2_coeff - A2_coeff * D1_coeff) / det;
b2 := -(A1_coeff * C2_coeff - A2_coeff * C1_coeff) / det;

// =======================================================================
// BƯỚC 3: Thay X0, Y0 vào phương trình mặt cầu 1 để tìm Z0
// Tạo thành phương trình bậc 2: A_quad * Z0^2 + B_quad * Z0 + C_quad = 0
// =======================================================================

A_quad := b1 * b1 + b2 * b2 + 1.0;
B_quad := 2.0 * (a1 * b1 + a2 * b2 - b2 * y_j1 - z_j1);
C_quad := a1 * a1 + a2 * a2 - 2.0 * a2 * y_j1 + r1 - (Forearm * Forearm);

// Tính Delta (Discriminant)
d := (B_quad * B_quad) - (4.0 * A_quad * C_quad);

// Kiểm tra xem vị trí các góc hiện tại có tạo ra tọa độ hợp lệ không
IF d < 0.0 THEN
    Calc_Forward_Kinematics := TRUE; // Trả về lỗi: Các khớp không thể kết nối
    RETURN;
END_IF;

// Tính tọa độ trung tâm End-Effector (Z lấy nghiệm có dấu trừ phía trước SQRT 
// vì đặc thù cơ cấu Delta robot làm việc ở nửa dưới trục Z)
OutZ := (-B_quad - SQRT(d)) / (2.0 * A_quad);

// Đẩy ngược Z0 vào hệ số tuyến tính để tìm X0 và Y0
OutX := a1 + b1 * OutZ;
OutY := a2 + b2 * OutZ;

Calc_OutZ := LREAL_TO_REAL(OutZ);
Calc_OutX := LREAL_TO_REAL(a1 + b1 * OutZ);
Calc_OutY := LREAL_TO_REAL(a2 + b2 * OutZ);

// Tính toán thành công
Calc_Forward_Kinematics := FALSE;
RETURN;
END_FUNCTION

FUNCTION_BLOCK MC_Home_Delta
VAR
    Move_Vel_Axis1 : MC_MoveVelocity;
    Start_Home : BOOL;
    MC_Stop_Axis1 : MC_Stop;
    Move_Vel_Axis2 : MC_MoveVelocity;
    Move_Vel_Axis3 : MC_MoveVelocity;
    MC_Stop_Axis2 : MC_Stop;
    MC_Stop_Axis3 : MC_Stop;
    MC_Home_Axis1 : MC_Home;
    MC_Home_Axis2 : MC_Home;
    MC_Home_Axis3 : MC_Home;
    t_home : TON;
    t2 : TON;
    t1 : TON;
    t3 : TON;
    TP1 : TP;
    TP2 : TP;
    TP4 : TP;
END_VAR
VAR_INPUT
    Start_Home_Ext : BOOL;
END_VAR
VAR_OUTPUT
    Done : BOOL;
END_VAR
VAR_EXTERNAL
    Home_Axis1 : BOOL;
    Home_Axis2 : BOOL;
    Home_Axis3 : BOOL;
END_VAR
VAR_EXTERNAL CONSTANT
    MC_Axis3 : _sAXIS_REF;
    MC_Axis2 : _sAXIS_REF;
    MC_Axis1 : _sAXIS_REF;
END_VAR
VAR_EXTERNAL
    Home_Lamp3 : BOOL;
    Home_Lamp1 : BOOL;
    Home_Lamp2 : BOOL;
    Start_Home_Flag : BOOL;
    Home_Done_Flag1 : BOOL;
    Home_Done_Flag2 : BOOL;
    Home_Done_Flag3 : BOOL;
END_VAR
VAR
    _e1 : R_TRIG;
    _e2 : R_TRIG;
    _e3 : R_TRIG;
    _e4 : R_TRIG;
END_VAR
(* ladder, written here as Structured Text *)

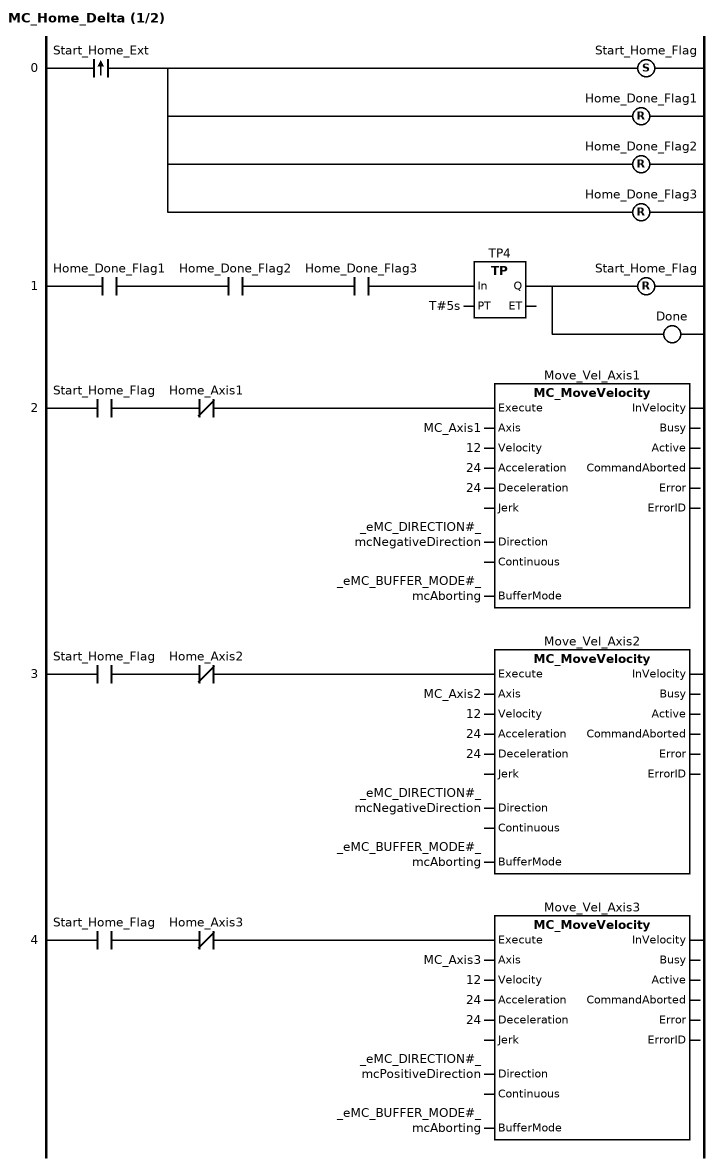
(* Rung 0 *)
_e1(CLK := Start_Home_Ext);
IF _e1.Q THEN
    Start_Home_Flag := TRUE;
    Home_Done_Flag1 := FALSE;
    Home_Done_Flag2 := FALSE;
    Home_Done_Flag3 := FALSE;
END_IF;
(* Rung 1 *)
TP4(In := Home_Done_Flag1 AND Home_Done_Flag2 AND Home_Done_Flag3, PT := T#5s);
IF TP4.Q THEN Start_Home_Flag := FALSE; END_IF;
Done := TP4.Q;
(* Rung 2 *)
Move_Vel_Axis1(Execute := Start_Home_Flag AND NOT Home_Axis1, Axis := MC_Axis1, Velocity := 12, Acceleration := 24, Deceleration := 24, Direction := _eMC_DIRECTION#_mcNegativeDirection, BufferMode := _eMC_BUFFER_MODE#_mcAborting);
(* Rung 3 *)
Move_Vel_Axis2(Execute := Start_Home_Flag AND NOT Home_Axis2, Axis := MC_Axis2, Velocity := 12, Acceleration := 24, Deceleration := 24, Direction := _eMC_DIRECTION#_mcNegativeDirection, BufferMode := _eMC_BUFFER_MODE#_mcAborting);
(* Rung 4 *)
Move_Vel_Axis3(Execute := Start_Home_Flag AND NOT Home_Axis3, Axis := MC_Axis3, Velocity := 12, Acceleration := 24, Deceleration := 24, Direction := _eMC_DIRECTION#_mcPositiveDirection, BufferMode := _eMC_BUFFER_MODE#_mcAborting);

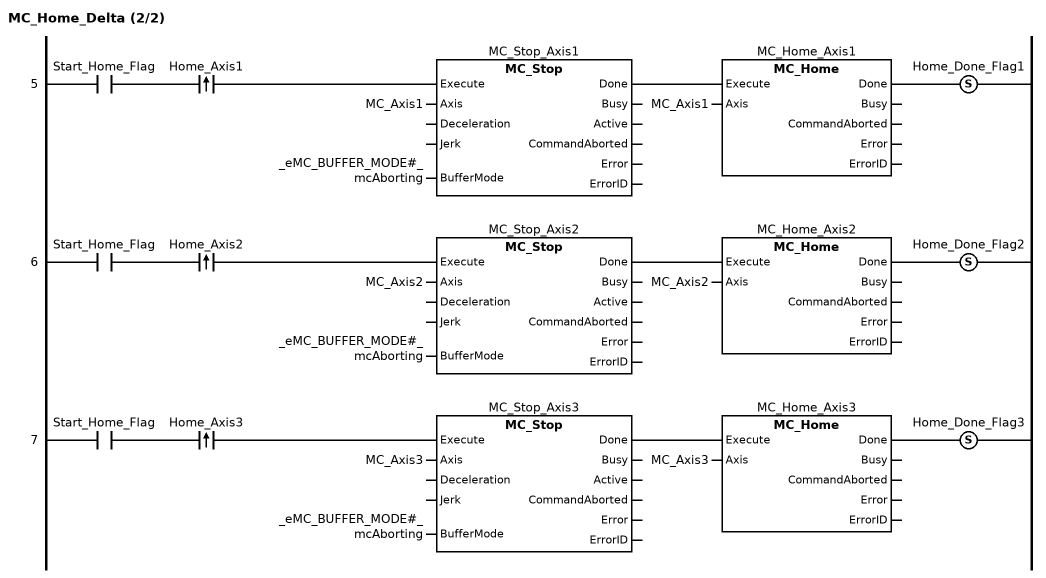
(* Rung 5 *)
_e2(CLK := Home_Axis1);
MC_Stop_Axis1(Execute := Start_Home_Flag AND _e2.Q, Axis := MC_Axis1, BufferMode := _eMC_BUFFER_MODE#_mcAborting);
MC_Home_Axis1(Execute := MC_Stop_Axis1.Done, Axis := MC_Axis1);
IF MC_Home_Axis1.Done THEN Home_Done_Flag1 := TRUE; END_IF;
(* Rung 6 *)
_e3(CLK := Home_Axis2);
MC_Stop_Axis2(Execute := Start_Home_Flag AND _e3.Q, Axis := MC_Axis2, BufferMode := _eMC_BUFFER_MODE#_mcAborting);
MC_Home_Axis2(Execute := MC_Stop_Axis2.Done, Axis := MC_Axis2);
IF MC_Home_Axis2.Done THEN Home_Done_Flag2 := TRUE; END_IF;
(* Rung 7 *)
_e4(CLK := Home_Axis3);
MC_Stop_Axis3(Execute := Start_Home_Flag AND _e4.Q, Axis := MC_Axis3, BufferMode := _eMC_BUFFER_MODE#_mcAborting);
MC_Home_Axis3(Execute := MC_Stop_Axis3.Done, Axis := MC_Axis3);
IF MC_Home_Axis3.Done THEN Home_Done_Flag3 := TRUE; END_IF;
END_FUNCTION_BLOCK

FUNCTION_BLOCK Goto_Absolute
VAR
    Out_Angle1 : LREAL;
    Out_Angle2 : LREAL;
    Out_Angle3 : LREAL;
    Move_abs0 : MC_MoveAbsolute;
    Move_abs1 : MC_MoveAbsolute;
    Move_abs2 : MC_MoveAbsolute;
END_VAR
VAR_INPUT
    Goto_Abs : BOOL;
    X_0 : LREAL;
    Y_0 : LREAL;
    Z_neg300 : LREAL;
END_VAR
VAR_OUTPUT
    Done : BOOL;
END_VAR
VAR_EXTERNAL CONSTANT
    MC_Axis1 : _sAXIS_REF;
    MC_Axis2 : _sAXIS_REF;
    MC_Axis3 : _sAXIS_REF;
END_VAR
VAR
    _t1 : BOOL;
    _e2 : F_TRIG;
END_VAR
(* ladder, written here as Structured Text *)

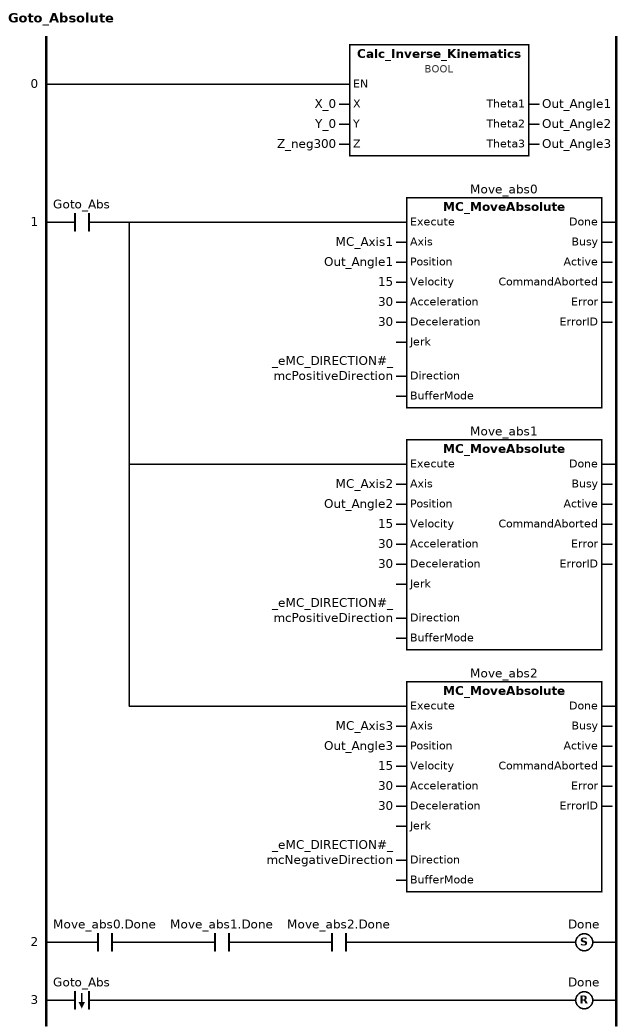
(* Rung 0 *)
_t1 := Calc_Inverse_Kinematics(X := X_0, Y := Y_0, Z := Z_neg300, Theta1 => Out_Angle1, Theta2 => Out_Angle2, Theta3 => Out_Angle3);
(* Rung 1 *)
Move_abs0(Execute := Goto_Abs, Axis := MC_Axis1, Position := Out_Angle1, Velocity := 15, Acceleration := 30, Deceleration := 30, Direction := _eMC_DIRECTION#_mcPositiveDirection);
Move_abs1(Execute := Goto_Abs, Axis := MC_Axis2, Position := Out_Angle2, Velocity := 15, Acceleration := 30, Deceleration := 30, Direction := _eMC_DIRECTION#_mcPositiveDirection);
Move_abs2(Execute := Goto_Abs, Axis := MC_Axis3, Position := Out_Angle3, Velocity := 15, Acceleration := 30, Deceleration := 30, Direction := _eMC_DIRECTION#_mcNegativeDirection);
(* Rung 2 *)
IF Move_abs0.Done AND Move_abs1.Done AND Move_abs2.Done THEN Done := TRUE; END_IF;
(* Rung 3 *)
_e2(CLK := Goto_Abs);
IF _e2.Q THEN Done := FALSE; END_IF;
END_FUNCTION_BLOCK

FUNCTION_BLOCK MC_Inter_Curve_Vel
VAR
    State : INT := 0;
    L : LREAL;
    t_acc : LREAL;
    t_dec : LREAL;
    S_acc : LREAL;
    S_dec : LREAL;
    S_run : LREAL;
    t_run : LREAL;
    T_total : LREAL;
    t : LREAL;
    t_phanh : LREAL;
    S_t : LREAL;
    X_t : LREAL;
    Y_t : LREAL;
    Z_t : LREAL;
    IK_Result : LREAL;
    Check_IK_Error : BOOL;
    tmp_Theta1 : LREAL;
    tmp_Theta2 : LREAL;
    tmp_Theta3 : LREAL;
    MC_Sync_Axis1 : MC_SyncMoveAbsolute;
    MC_Sync_Axis2 : MC_SyncMoveAbsolute;
    MC_Sync_Axis3 : MC_SyncMoveAbsolute;
    Actual_Vmax : LREAL := 100;
    tau : LREAL := 0.2;
    Init_Counter : INT;
    Target_Theta1 : LREAL;
    Target_Theta2 : LREAL;
    Target_Theta3 : LREAL;
    Start_Theta1 : LREAL;
    Start_Theta2 : LREAL;
    Start_Theta3 : LREAL;
    cycle_count : INT;
    Enable_Motion : BOOL;
    MC_SyncMoveAbsolute_Axis1 : MC_SyncMoveAbsolute;
    MC_SyncMoveAbsolute_Axis2 : MC_SyncMoveAbsolute;
    MC_SyncMoveAbsolute_Axis3 : MC_SyncMoveAbsolute;
    Use_Standard_SCurve : BOOL;
    S_limit : LREAL;
    V_reach : LREAL;
    Vec1_X : LREAL;
    Vec1_Y : LREAL;
    Vec1_Z : LREAL;
    Vec2_X : LREAL;
    Vec2_Y : LREAL;
    Vec2_Z : LREAL;
    Len1 : LREAL;
    Len2 : LREAL;
    Cos_Theta : LREAL;
    V_Corner_Max : LREAL;
END_VAR
VAR_INPUT
    X_A : LREAL;
    Y_A : LREAL;
    Z_A : LREAL;
    X_B : LREAL;
    Y_B : LREAL;
    Z_B : LREAL;
    V_max : LREAL;
    A_max : LREAL;
    D_max : LREAL;
END_VAR
VAR_OUTPUT
    Theta1 : LREAL;
    Theta2 : LREAL;
    Theta3 : LREAL;
    Out_Error_IK_OWS : BOOL;
    Done : BOOL;
    Busy : BOOL;
END_VAR
VAR_INPUT
    V_Start_Req : LREAL;
END_VAR
VAR_OUTPUT
    Out_Done_Inter : BOOL;
    Out_Done_Blend : BOOL;
    Out_V_End : LREAL;
END_VAR
VAR_INPUT
    Why : BOOL;
    Blend_mode : BOOL;
END_VAR
VAR_IN_OUT
    Execute : BOOL;
END_VAR
VAR_OUTPUT
    t_total_estimate : LREAL;
END_VAR
VAR_INPUT
    X_C : LREAL;
    Y_C : LREAL;
    Z_C : LREAL;
END_VAR
VAR_OUTPUT
    ICV_t5_out : LREAL;
END_VAR
VAR_EXTERNAL CONSTANT
    MC_Axis2 : _sAXIS_REF;
    MC_Axis3 : _sAXIS_REF;
    MC_Axis1 : _sAXIS_REF;
END_VAR
// ====================================================================
// PHẦN 1: TÍNH TOÁN QUỸ ĐẠO BÊN TRONG STATE MACHINE
// ====================================================================
CASE State OF
    0:  // ================= Step 0: waiting for the new command =================
        IF Execute = TRUE THEN
            Out_Error_IK_OWS := FALSE;  // Reset all fault
            Out_Done_Inter := FALSE;  // Reset interpolation flag
            
            // Cal the inverse kinematic for check the valid of the point
            Check_IK_Error := calc_inverse_kinematics(
                X := X_A, Y := Y_A, Z := Z_A, 
                Theta1 => Target_Theta1, Theta2 => Target_Theta2, Theta3 => Target_Theta3
            );
            
            IF Check_IK_Error = TRUE THEN
                Out_Error_IK_OWS := TRUE; 
                State := 99; 
            ELSE
                Enable_Motion := TRUE;  
                
                // LỰA CHỌN LOGIC XUẤT PHÁT DỰA VÀO VẬN TỐC ĐẦU VÀO
                IF V_Start_Req > 0.0 THEN
                    // ĐANG CHẠY NỐI TIẾP (Blend): 
                    // Bỏ qua State 10 làm mượt. Dùng luôn góc lý thuyết Target làm xuất phát để tránh giật
                    Theta1 := Target_Theta1;
                    Theta2 := Target_Theta2;
                    Theta3 := Target_Theta3;
                    State := 1; // Chuyển thẳng sang tính toán S-Curve
                ELSE
                    // XUẤT PHÁT TỪ TRẠNG THÁI DỪNG HẲN: 
                    // Phải lấy vị trí thực tế Act.Pos để chạy mượt 20 chu kỳ triệt tiêu sai số
                    Start_Theta1 := MC_Axis1.Act.Pos; 
                    Start_Theta2 := MC_Axis2.Act.Pos;
                    Start_Theta3 := MC_Axis3.Act.Pos;
                    cycle_count := 1;
                    State := 10; 
                END_IF;
            END_IF;
        ELSE
            // KHI EXECUTE = FALSE
            // Ngắt cờ Blend thành dạng xung (Pulse) để Main Program bắt tín hiệu
            Out_Done_Blend := FALSE; 
            
            Enable_Motion := FALSE; 
            Theta1 := MC_Axis1.Act.Pos;
            Theta2 := MC_Axis2.Act.Pos;
            Theta3 := MC_Axis3.Act.Pos;
        END_IF;

    10: (*
    // =====Step 10: smothing the point start and actual point (from servo) with 20 cyclic time=======
    *)
        IF cycle_count <= 20 THEN
            Theta1 := Start_Theta1 + (Target_Theta1 - Start_Theta1) * (INT_TO_REAL(cycle_count) / 20.0);
            Theta2 := Start_Theta2 + (Target_Theta2 - Start_Theta2) * (INT_TO_REAL(cycle_count) / 20.0);
            Theta3 := Start_Theta3 + (Target_Theta3 - Start_Theta3) * (INT_TO_REAL(cycle_count) / 20.0);
            cycle_count := cycle_count + 1;
        ELSE
            State := 1;
        END_IF;

    1:  // ================= BƯỚC 1: TÍNH TOÁN CẤU HÌNH ĐỘNG LỰC HỌC (S-CURVE/TRAPEZOIDAL) =================
        L := SQRT((X_B - X_A)**2 + (Y_B - Y_A)**2 + (Z_B - Z_A)**2); 

        IF L > 0.0 THEN
            IF Blend_Mode = FALSE THEN
                // --- TRƯỜNG HỢP 1: LÀ ĐIỂM CUỐI CÙNG -> TỰ ĐỘNG PHANH VỀ 0 ---
                Out_V_End := 0.0;
                Use_Standard_SCurve := (V_Start_Req = 0.0); 
                Actual_Vmax := V_max;

                IF Use_Standard_SCurve = TRUE THEN
                    IF L < (0.75 * (Actual_Vmax**2) * (1.0/A_max + 1.0/D_max)) THEN
                        Actual_Vmax := SQRT(L / (0.75 * (1.0/A_max + 1.0/D_max)));
                    END_IF;

                    t_acc := 1.5 * (Actual_Vmax / A_max);
                    t_dec := 1.5 * (Actual_Vmax / D_max);
                    S_acc := 0.5 * Actual_Vmax * t_acc;
                    S_dec := 0.5 * Actual_Vmax * t_dec;
                    S_run := L - S_acc - S_dec;
                    t_run := S_run / Actual_Vmax;
                    T_total := t_acc + t_run + t_dec;
                ELSE
                    S_limit := (ABS(Actual_Vmax**2 - V_Start_Req**2)/(2.0*A_max)) + (ABS(Actual_Vmax**2)/(2.0*D_max));
                    IF S_limit > L THEN
                        Actual_Vmax := SQRT((2.0*A_max*D_max*L + D_max*(V_Start_Req**2)) / (A_max + D_max));
                    END_IF;

                    t_acc := ABS(Actual_Vmax - V_Start_Req) / A_max;
                    t_dec := ABS(Actual_Vmax) / D_max; 
                    S_acc := (V_Start_Req + Actual_Vmax) * 0.5 * t_acc;
                    S_dec := Actual_Vmax * 0.5 * t_dec;
                    S_run := L - S_acc - S_dec;
                    
                    IF S_run < 0.0 THEN S_run := 0.0; END_IF;
                    t_run := S_run / Actual_Vmax;
                    T_total := t_acc + t_run + t_dec;
                END_IF;

            ELSE
                // --- TRƯỜNG HỢP 2: CHẠY NỐI TIẾP (BLEND) CÓ TÍNH TOÁN LOOK-AHEAD GÓC CUA ---
                Use_Standard_SCurve := FALSE;
                
                // 1. Tính toán 2 Vector để xác định góc rẽ tại B
                Vec1_X := X_B - X_A; Vec1_Y := Y_B - Y_A; Vec1_Z := Z_B - Z_A;
                Vec2_X := X_C - X_B; Vec2_Y := Y_C - Y_B; Vec2_Z := Z_C - Z_B;
                
                Len1 := L; 
                Len2 := SQRT(Vec2_X**2 + Vec2_Y**2 + Vec2_Z**2); 
                
                // 2. Tính Cosin của góc lệch (Cos_Theta)
                IF (Len1 > 0.0) AND (Len2 > 0.0) THEN
                    Cos_Theta := (Vec1_X*Vec2_X + Vec1_Y*Vec2_Y + Vec1_Z*Vec2_Z) / (Len1 * Len2);
                    // Ép kiểu an toàn tránh lỗi dấu phẩy động (NaN) của PLC
                    IF Cos_Theta > 1.0 THEN Cos_Theta := 1.0; ELSIF Cos_Theta < -1.0 THEN Cos_Theta := -1.0; END_IF;
                ELSE
                    Cos_Theta := 1.0; // Đi thẳng nếu 2 điểm vô tình trùng nhau
                END_IF;

                // 3. Quy đổi góc ra giới hạn vận tốc an toàn tại góc cua
                V_Corner_Max := V_max * SQRT((Cos_Theta + 1.0) / 2.0);

                // 4. Kiểm tra vận tốc dự phóng và chốt Vận tốc cuối (Out_V_End)
                V_reach := SQRT(V_Start_Req**2 + 2.0 * A_max * L);
                
                Out_V_End := V_Corner_Max;
                IF Out_V_End > V_reach THEN Out_V_End := V_reach; END_IF;
                IF Out_V_End > V_max THEN Out_V_End := V_max; END_IF;

                // 5. Tính toán cấu hình hình thang (Tăng tốc - Chạy đều - Giảm tốc vào cua)
                Actual_Vmax := V_max;
                S_limit := (ABS(Actual_Vmax**2 - V_Start_Req**2)/(2.0*A_max)) + (ABS(Actual_Vmax**2 - Out_V_End**2)/(2.0*D_max));

                IF S_limit > L THEN
                    // Không đủ quãng đường để đạt V_max, tạo Profile hình tam giác chóp
                    Actual_Vmax := SQRT((2.0*A_max*D_max*L + D_max*(V_Start_Req**2) + A_max*(Out_V_End**2)) / (A_max + D_max));
                END_IF;

                // Safety Clamp: Đảm bảo sai số làm tròn không khiến Actual_Vmax nhỏ hơn các điểm mút
                IF Actual_Vmax < V_Start_Req THEN Actual_Vmax := V_Start_Req; END_IF;
                IF Actual_Vmax < Out_V_End THEN Actual_Vmax := Out_V_End; END_IF;

                t_acc := ABS(Actual_Vmax - V_Start_Req) / A_max;
                t_dec := ABS(Actual_Vmax - Out_V_End) / D_max; 
                
                S_acc := (V_Start_Req + Actual_Vmax) * 0.5 * t_acc;
                S_dec := (Out_V_End + Actual_Vmax) * 0.5 * t_dec;
                S_run := L - S_acc - S_dec;
                
                IF S_run < 0.0 THEN S_run := 0.0; END_IF;
                t_run := S_run / Actual_Vmax;
                T_total := t_acc + t_run + t_dec;
            END_IF;

            // ====================================================================
            // TÍNH TOÁN t_total_estimate BAO GỒM MỌI TRƯỜNG HỢP
            // ====================================================================
            IF V_Start_Req = 0.0 THEN
                t_total_estimate := T_total + 0.08; // Cộng thêm 20 chu kỳ (0.08s) của State 10
            ELSE
                t_total_estimate := T_total;
            END_IF;
            ICV_t5_out := t_total_estimate;
            t := 0.0;     
            State := 2;   
        ELSE
            Execute := FALSE;
            State := 0;
        END_IF;

    2:  // ================= BƯỚC 2: NỘI SUY TỌA ĐỘ THEO THỜI GIAN =================
        IF t <= T_total THEN
            // 2.1 Tính quãng đường S_t
            IF Use_Standard_SCurve = TRUE THEN
                IF t <= t_acc THEN
                    tau := t / t_acc; 
                    S_t := Actual_Vmax * t_acc * ((tau ** 3) - 0.5 * (tau ** 4));
                ELSIF t <= (t_acc + t_run) THEN
                    S_t := S_acc + Actual_Vmax * (t - t_acc);
                ELSE
                    t_phanh := t - (t_acc + t_run);
                    tau := t_phanh / t_dec; 
                    S_t := S_acc + S_run + Actual_Vmax * t_dec * (tau - (tau ** 3) + 0.5 * (tau ** 4));
                END_IF;
            ELSE
                IF t <= t_acc THEN
                    S_t := V_Start_Req * t + 0.5 * A_max * (t**2);
                ELSIF t <= (t_acc + t_run) THEN
                    S_t := S_acc + Actual_Vmax * (t - t_acc);
                ELSE
                    t_phanh := t - (t_acc + t_run);
                    S_t := S_acc + S_run + Actual_Vmax * t_phanh - 0.5 * D_max * (t_phanh**2);
                END_IF;
                
                IF S_t > L THEN S_t := L; END_IF; 
            END_IF;

            // 2.2 Tính tọa độ Descartes X, Y, Z tại S_t
            X_t := X_A + (S_t / L) * (X_B - X_A);
            Y_t := Y_A + (S_t / L) * (Y_B - Y_A);
            Z_t := Z_A + (S_t / L) * (Z_B - Z_A);

            // 2.3 Giải Động Học Nghịch (IK) để tìm góc cho 3 trục
            Check_IK_Error := calc_inverse_kinematics(
                X := X_t, Y := Y_t, Z := Z_t, 
                Theta1 => tmp_Theta1, Theta2 => tmp_Theta2, Theta3 => tmp_Theta3
            );
            
            IF Check_IK_Error = TRUE THEN
                Out_Error_IK_OWS := TRUE; 
                State := 99; 
                RETURN; 
            END_IF;

            // Cập nhật vị trí đẩy xuống lệnh gọi Servo
            Theta1 := tmp_Theta1;
            Theta2 := tmp_Theta2;
            Theta3 := tmp_Theta3;

            t := t + 0.004; // Chu kỳ lấy mẫu nội suy (4ms)

        ELSE
            // ================= KẾT THÚC ĐOẠN ĐƯỜNG (HẾT THỜI GIAN T_total) =================
            IF (Blend_Mode = TRUE) AND (Out_V_End > 0.0) THEN
                // CHẠY NỐI TIẾP: Bật cờ Blend, chờ nhả Execute
                Out_Done_Blend := TRUE; 
                Execute := FALSE; 
                State := 0; // Quay về State 0 chực chờ nạp điểm mới và nội suy tiếp
            ELSE
                // DỪNG HẲN: Chuyển sang State 3 đợi Servo Settle
                State := 3; 
            END_IF;
        END_IF;

    3:  // ================= BƯỚC 3: KIỂM TRA SAI SỐ DỪNG (SETTLE) =================
        Enable_Motion := FALSE; 
        
        // Đọc ACT.POS để xác nhận Servo đã bám sát điểm đích với sai số < 0.0005 độ
        IF (ABS(Theta1 - MC_Axis1.Act.Pos) <= 0.0005) AND 
           (ABS(Theta2 - MC_Axis2.Act.Pos) <= 0.0005) AND 
           (ABS(Theta3 - MC_Axis3.Act.Pos) <= 0.0005)
           THEN
            Out_Done_Inter := TRUE;
        ELSE
            Out_Done_Inter := FALSE;
        END_IF;

        // Xả cờ và reset State khi Servo báo hết Busy
        IF (MC_Sync_Axis1.Busy = FALSE) AND 
           (MC_Sync_Axis2.Busy = FALSE) AND 
           (MC_Sync_Axis3.Busy = FALSE) THEN
            
            Execute := FALSE;  
            State := 0;        
        END_IF;

    99: // ================= BƯỚC 99: LỖI KINEMATICS =================
        Execute := FALSE;
        Enable_Motion := FALSE; 
        IF Out_Error_IK_OWS = FALSE THEN
             State := 0;
        END_IF;
END_CASE;

// ====================================================================
// PHẦN 2: GỌI HÀM SERVO (LUÔN ĐƯỢC QUÉT Ở CUỐI CHU KỲ)
// ====================================================================
// Sử dụng hàm đồng bộ vị trí, servo sẽ bám theo biến Theta liên tục
MC_Sync_Axis1(Axis := MC_Axis1, Execute := Enable_Motion, Position := Theta1);
MC_Sync_Axis2(Axis := MC_Axis2, Execute := Enable_Motion, Position := Theta2);
MC_Sync_Axis3(Axis := MC_Axis3, Execute := Enable_Motion, Position := Theta3);
END_FUNCTION_BLOCK